ABB RobotStudio station: burguerBotVentosaYCintaDef2.rspag

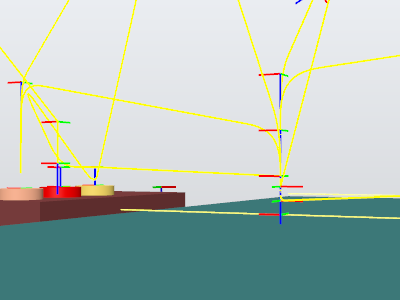
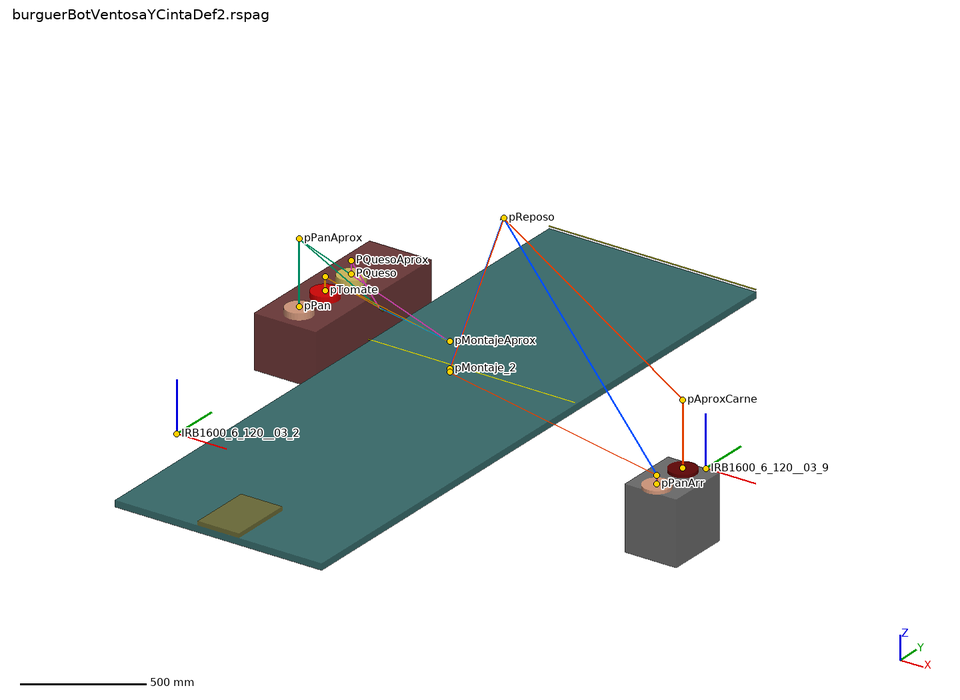
[picture v1: parts stored in the station drawn from their meshes, with robot base, taught points and paths (robot models come from the ABB library and are not in the file)]
--- station ---
Station Station (saved by RobotStudio 24.1.10713.1)
Controller Controlador2, task T_ROB1: task frame (RAPID world) sits at (2496.48, 947.06, 0) mm, rotated rx 0 ry 0 rz 179.92 deg in the station
Controller Controlador4, task T_ROB1: task frame (RAPID world) sits at (600, 0, 0) mm in the station
Controller Controlador4
  mechanical unit ROB_1: IRB1600_6_120__03_2, 6 joints, base frame (0, 0, 0) mm
Controller Controlador2
  mechanical unit ROB_1: IRB1600_6_120__03_9, 6 joints, base frame (0, 0, 0) mm
Layout (positions relative to the parent item):
  - Ventosa [mechanism, from Libraries\Ventosa.rslib] at (1406.29, 0, 929) mm, rotated rx 180 ry 60 rz 180 deg
  - CintaTransportadora [part] at (0, 0, -530) mm, size 1000 x 3000 x 30 mm
  - IRB1600_6_120__03_2 [mechanism, from %ABB.RobotStudio.Models.IRB1600%\IRB1600_6_120_G_03.rslib] at (600, 0, 0) mm; joint values [0, 0, 0, 0, 0.5236, 0] (rad or m)
  - SmartComponent_2 [smart component]
      signals: DO PiezaDetectada, DI ActivaVentosa, DO Vacuostato
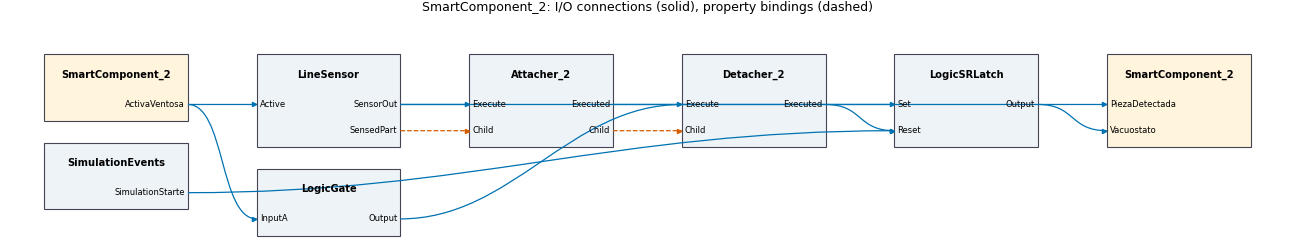
      connections:
        SmartComponent_2.ActivaVentosa -> LineSensor.Active
        SmartComponent_2.ActivaVentosa -> LogicGate.InputA
        LogicGate.Output -> Detacher_2.Execute
        LineSensor.SensorOut -> Attacher_2.Execute
        LineSensor.SensorOut -> SmartComponent_2.PiezaDetectada
        Attacher_2.Executed -> LogicSRLatch.Set
        Detacher_2.Executed -> LogicSRLatch.Reset
        SimulationEvents.SimulationStarted -> LogicSRLatch.Reset
        LogicSRLatch.Output -> SmartComponent_2.Vacuostato
        Attacher_2.Child => Detacher_2.Child
        LineSensor.SensedPart => Attacher_2.Child
    - LineSensor [smart component, from Components\LineSensor.rslib] at (1579.5, 0, 829) mm, rotated rx 180 ry 60 rz 180 deg
        properties: Start=[0 0 -0.002]; End=[0 0 0.02]; Length=0.022; Radius=0.002; Tag=(none); SensedPart=(none); SensedPoint=[0 0 0]
      - _sensorPart_ [part], size 4 x 4 x 22 mm
    - SimulationEvents [smart component, from Components\SimulationEvents.rslib]
    - LogicSRLatch [smart component, from Components\LogicSRLatch.rslib]
    - Attacher_2 [smart component, from Components\Attacher.rslib]
        properties: Parent=Ventosa; Flange=0; Child=(none); Mount=false; Offset=[0 0 0]; Orientation=[0 0 0]
    - Detacher_2 [smart component, from Components\Detacher.rslib]
        properties: Child=(none); KeepPosition=true
    - LogicGate [smart component, from Components\LogicGate.rslib]
        properties: Operator=NOT; Delay=0
  - Pieza_3 [part], size 1050 x 3000 x 100 mm
  - Pieza_7 [part] at (0, -1450, -30) mm, size 200 x 300 x 20 mm
  - SmartComponent_3 [smart component] at (0, 0, -530) mm
      signals: DI PideNuevaPieza, DI MueveCinta, DI Desencolar, DO Hamburguesa_detectada
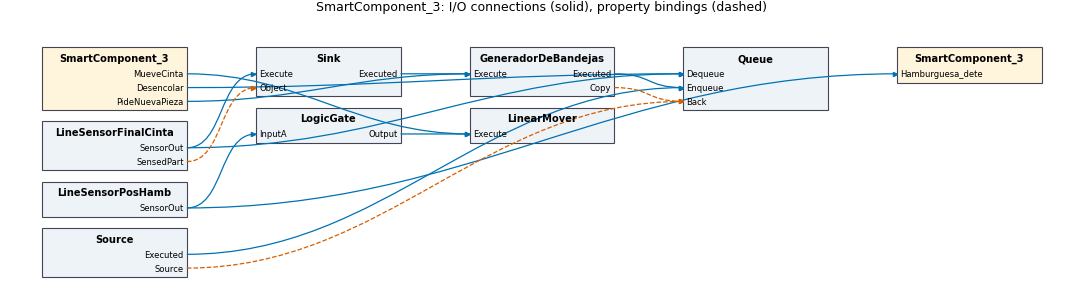
      connections:
        SmartComponent_3.MueveCinta -> LinearMover.Execute
        SmartComponent_3.Desencolar -> Queue.Dequeue
        SmartComponent_3.PideNuevaPieza -> GeneradorDeBandejas.Execute
        GeneradorDeBandejas.Executed -> Queue.Enqueue
        Sink.Executed -> GeneradorDeBandejas.Execute
        LineSensorFinalCinta.SensorOut -> Sink.Execute
        LineSensorFinalCinta.SensorOut -> Queue.Dequeue
        LineSensorPosHamb.SensorOut -> LogicGate.InputA
        LogicGate.Output -> LinearMover.Execute
        LineSensorPosHamb.SensorOut -> SmartComponent_3.Hamburguesa_detectada
        Source.Executed -> Queue.Enqueue
        GeneradorDeBandejas.Copy => Queue.Back
        LineSensorFinalCinta.SensedPart => Sink.Object
        Source.Source => Queue.Back
    - GeneradorDeBandejas [smart component, from Components\Source.rslib]
        properties: Source=Pieza_7; Copy=(none); Parent=(none); Position=[0 -1.45 -0.03]; Orientation=[0 0 0]; Transient=false; PhysicsBehavior=-1
    - LinearMover [smart component, from Components\LinearMover.rslib]
        properties: Object=Queue; Direction=[0 1 0]; Speed=0.2; Reference=Global; ReferenceObject=(none)
    - Queue [smart component, from Components\Queue.rslib]
        properties: Back=(none); Front=(none); Queue={1fa18e9d-088c-41fe-8e63-321db63f1bad};{66fc0b19-5291-4fa8-960b-30c1fd8ad654};{bf5ac1da-f569-4681-bc2f-d1bebfeb1945};{a7c02364-1145-4610-8c2b-21e8e4e74e7e};{e07134d1-5b8f-4729-998b-d35f37be9415};{77c18e64-ed22-4101-8412-22759ad2fd65};{e3f1d31c-383c-4d57-a647-59baedf5051e};{31de0638-30c3-4a0d-b96c-771df3fa9e8e};{ccf4f79c-bd7e-444b-aa3a-f3a101a5e061};{9c3ce438-0d0a-462d-859f-6c1952ce2779};{2c210c3e-426b-4bc3-92f0-a2b14ac0cff1};{860f6b89-5f7b-417f-be90-2e5516634339};{3c4b279c-e194-41e7-8d5b-6c695006562c};{9a04805c-3299-4768-adf6-effe421ff297};{2ba32a07-e99c-497b-b6b1-776f4c664f37};{e5d152f1-81eb-4789-a107-4ce79efd876e};{84050f51-b700-43f5-9d48-1de7078c80f2};{da5c4f3e-e2de-4859-8c8b-22e5639c2eb3};{b8627b52-6deb-4d66-bbe9-42a0777c5345};{afe129ed-1453-4d5a-b210-b8758cc1c2e1};{660fbeab-b469-451a-a4fe-b26f68304c6b};{d46f86e2-3b48-4b92-a915-6ed2dcae6b65};{75fa054e-13a5-4b2b-a626-0fa9227d0997};{dc2c9636-b798-4d71-ba5e-8e763e159b99};{52b1206f-a2cb-4ff9-8ba0-982d9823dc0e};{f684843b-9464-44eb-8d71-6faa8fd13188};{26aecd76-d99c-4597-b4e3-adbf34ae068a};{1ac82643-5105-46b1-9dd2-ef4d0df968c2}; NumberOfObjects=2
    - Sink [smart component, from Components\Sink.rslib]
        properties: Object=(none)
    - LineSensorFinalCinta [smart component, from Components\LineSensor.rslib]
        properties: Start=[2 2 0.76]; End=[1 2 0.76]; Length=1; Radius=0.002; Tag=(none); SensedPart=(none); SensedPoint=[0 0 0]
      - _sensorPart_ [part], size 1000 x 4 x 4 mm
    - LineSensorPosHamb [smart component, from Components\LineSensor.rslib]
        properties: Start=[2 0.75 0.76]; End=[1 0.75 0.76]; Length=1; Radius=0.002; Tag=(none); SensedPart=(none); SensedPoint=[0 0 0]
      - _sensorPart_ [part], size 1000 x 4 x 4 mm
    - LogicGate [smart component, from Components\LogicGate.rslib]
        properties: Operator=NOT; Delay=0
    - Source [smart component, from Components\Source.rslib]
        properties: Source=Pan2; Copy=(none); Parent=(none); Position=[0 0 0]; Orientation=[0 0 0]; Transient=false; PhysicsBehavior=-1
  - Ventosa_2 [mechanism, from Libraries\Ventosa.rslib] at (1690.19, 948.21, 929) mm, rotated rx -180 ry 60 rz -0.08 deg
  - SmartComponent_4 [smart component]
      signals: DO PiezaDetectada, DO Vacuostato, DI ActivaVentosa2
      connections:
        LogicGate.Output -> Detacher_2.Execute
        LineSensor.SensorOut -> Attacher_2.Execute
        LineSensor.SensorOut -> SmartComponent_4.PiezaDetectada
        Attacher_2.Executed -> LogicSRLatch.Set
        Detacher_2.Executed -> LogicSRLatch.Reset
        SimulationEvents.SimulationStarted -> LogicSRLatch.Reset
        LogicSRLatch.Output -> SmartComponent_4.Vacuostato
        SmartComponent_4.ActivaVentosa2 -> LineSensor.Active
        SmartComponent_4.ActivaVentosa2 -> LogicGate.InputA
        Attacher_2.Child => Detacher_2.Child
        LineSensor.SensedPart => Attacher_2.Child
    - LineSensor [smart component, from Components\LineSensor.rslib] at (1516.99, 948.46, 829) mm, rotated rx -180 ry 60 rz -0.08 deg
        properties: Start=[0 0 -0.002]; End=[0 0 0.02]; Length=0.022; Radius=0.002; Tag=(none); SensedPart=(none); SensedPoint=[0 0 0]
      - _sensorPart_ [part], size 4 x 4 x 22 mm
    - SimulationEvents [smart component, from Components\SimulationEvents.rslib]
    - LogicSRLatch [smart component, from Components\LogicSRLatch.rslib]
    - Attacher_2 [smart component, from Components\Attacher.rslib]
        properties: Parent=Ventosa_2; Flange=0; Child=(none); Mount=false; Offset=[0 0 0]; Orientation=[0 0 0]
    - Detacher_2 [smart component, from Components\Detacher.rslib]
        properties: Child=(none); KeepPosition=true
    - LogicGate [smart component, from Components\LogicGate.rslib]
        properties: Operator=NOT; Delay=0
  - Pieza_11 [part], size 304.8 x 406.3 x 254 mm
  - Pieza_12 [part], size 125 x 124.3 x 30 mm
  - Pieza_14 [part], size 250 x 300 x 300 mm
  - Pieza_15 [part] at (0, 75, 0) mm, size 125 x 124.3 x 15 mm
  - IRB1600_6_120__03_9 [mechanism, from %ABB.RobotStudio.Models.IRB1600%\IRB1600_6_120_G_03.rslib] at (2496.48, 947.06, 0) mm, rotated rx 0 ry 0 rz 179.92 deg; joint values [0, 0, 0, 0, 0.5236, 0] (rad or m)
  - Tomate [part] at (0, 180, 0) mm, size 125 x 124.3 x 30 mm
  - Queso [part] at (0, 360, 0) mm, size 125 x 124.3 x 30 mm
  - Pan2 [part] at (0, -105, 0) mm, size 125 x 124.3 x 15 mm
  - Pieza_18 [part] at (0, 400, 0) mm, size 300 x 400 x 250 mm
  - Pieza_7_11 [part] at (0, -1450, -30) mm, size 200 x 300 x 20 mm
  - Pieza_7_51 [part] at (0, -1450, -30) mm, size 200 x 300 x 20 mm
  - Pieza_7_54 [part] at (0, -1450, -30) mm, size 200 x 300 x 20 mm
  - Pieza_7_2 [part] at (0, -1450, -30) mm, size 200 x 300 x 20 mm
Attachment: Ventosa is attached to IRB1600_6_120__03_2 / Link6
Attachment: LineSensor is attached to Ventosa / PiezaVentosa
Attachment: SmartComponent_3 is attached to CintaTransportadora
Attachment: LineSensor is attached to Ventosa_2 / PiezaVentosa
Attachment: Ventosa_2 is attached to IRB1600_6_120__03_9 / Link6
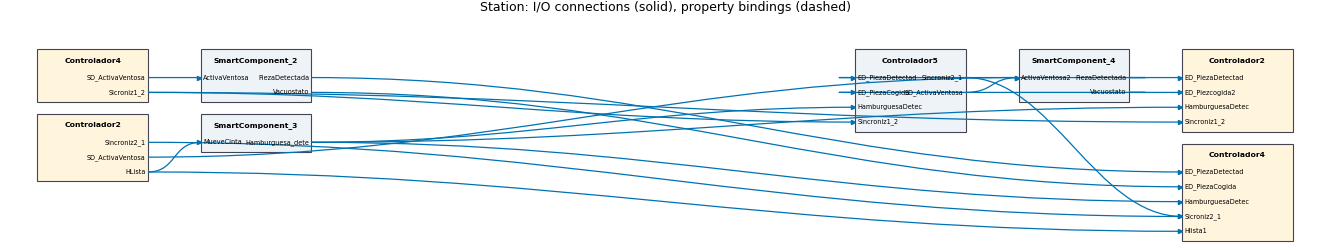
Station logic (signal -> signal, property => property):
  SmartComponent_2.PiezaDetectada -> Controlador4.ED_PiezaDetectada
  Controlador4.SD_ActivaVentosa -> SmartComponent_2.ActivaVentosa
  SmartComponent_2.Vacuostato -> Controlador4.ED_PiezaCogida
  SmartComponent_3.Hamburguesa_detectada -> Controlador4.HamburguesaDetect
  SmartComponent_4.PiezaDetectada -> Controlador5.ED_PiezaDetectada
  SmartComponent_4.Vacuostato -> Controlador5.ED_PiezaCogida
  SmartComponent_3.Hamburguesa_detectada -> Controlador5.HamburguesaDetect
  Controlador5.Sincroniz2_1 -> Controlador4.Sicroniz2_1
  Controlador4.Sicroniz1_2 -> Controlador5.Sincroniz1_2
  SmartComponent_4.PiezaDetectada -> Controlador2.ED_PiezaDetectada2
  SmartComponent_4.Vacuostato -> Controlador2.ED_Piezcogida2
  SmartComponent_3.Hamburguesa_detectada -> Controlador2.HamburguesaDetect2
  Controlador4.Sicroniz1_2 -> Controlador2.Sincroniz1_2
  Controlador2.Sincroniz2_1 -> Controlador4.Sicroniz2_1
  ?.SD_ActivaVentosa -> SmartComponent_4.ActivaVentosa2
  Controlador2.SD_ActivaVentosa -> SmartComponent_4.ActivaVentosa2
  Controlador2.HLista -> SmartComponent_3.MueveCinta
  Controlador2.HLista -> Controlador4.Hlista1

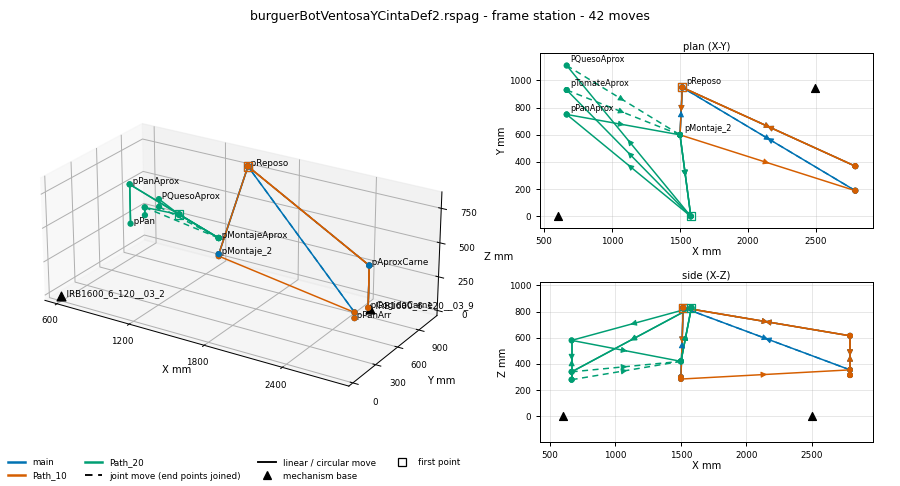
[picture p0: tool path of burguerBotVentosaYCintaDef2.rspag in frame station, 42 of 47 moves have a stored position in this frame; points joined in program order, loops and branches not executed]
--- Backups/Controlador2/RAPID/TASK1/PROGMOD/CalibData.mod ---
MODULE CalibData
    PERS tooldata Ventosa:=[TRUE,[[0,0,200],[1,0,0,0]],[1,[0,0,125],[1,0,0,0],0.002,0.002,0.0013]];
ENDMODULE

--- Backups/Controlador2/RAPID/TASK1/PROGMOD/Module1.mod ---
MODULE Module1
    CONST robtarget pReposo:=[[979.496732003,0,829],[0.5,0,0.866025404,0],[0,0,-1,0],[9E+09,9E+09,9E+09,9E+09,9E+09,9E+09]];
    CONST robtarget pAproxCarne:=[[-294.1282673,577.734595344,615],[0,0.999999744,0.000716141,0],[1,0,1,0],[9E+09,9E+09,9E+09,9E+09,9E+09,9E+09]];
    CONST robtarget pCogidaCarne:=[[-294.1282673,577.734595344,315],[0,0.999999744,0.000716141,0],[1,0,1,0],[9E+09,9E+09,9E+09,9E+09,9E+09,9E+09]];
    CONST robtarget pMontaje_2:=[[995.982835611,348.8831626,300],[0,-0.000716141,0.999999744,0],[0,0,0,0],[9E+09,9E+09,9E+09,9E+09,9E+09,9E+09]];
    CONST robtarget pMontaje:=[[995.982835611,348.8831626,285],[0,-0.000716141,0.999999744,0],[0,0,0,0],[9E+09,9E+09,9E+09,9E+09,9E+09,9E+09]];
    CONST robtarget pPanArr_2:=[[-294.386077932,757.734410716,355],[0,0.999999744,0.000716141,0],[1,0,-1,0],[9E+09,9E+09,9E+09,9E+09,9E+09,9E+09]];
    CONST robtarget pPanArr:=[[-294.386077932,757.734410716,315],[0,0.999999744,0.000716141,0],[1,0,-1,0],[9E+09,9E+09,9E+09,9E+09,9E+09,9E+09]];
!***********************************************************
    !
    ! M?dulo:  Module1
    !
    ! Descripción:
    !   <Introduzca la descripción aquí>
    !
    ! Autor: rafac
    !
    ! Versión: 1.0
    !
    !***********************************************************


    !***********************************************************
    !
    ! Procedimiento Main
    !
    !   Este es el punto de entrada de su programa
    !
    !***********************************************************
    PROC main()
        VAR robtarget aux;
        SetDO Sincroniz2_1,0;
        SetDO HLista, 0;
         WaitDI Sincroniz1_2,1;
            MoveL pReposo,v1000,z100,Ventosa\WObj:=wobj0;
            MoveJ pAproxCarne,v1000,fine,Ventosa\WObj:=wobj0;
            MoveL pCogidaCarne,v500,fine,Ventosa\WObj:=wobj0;
            SetDO SD_ActivaVentosa,1;
            WaitDI ED_Piezcogida2,1;

            MoveL pAproxCarne,v1000,fine,Ventosa\WObj:=wobj0;
            MoveJ pReposo,v1000,fine,Ventosa\WObj:=wobj0;

            MoveL pMontaje_2,v1000,fine,Ventosa\WObj:=wobj0;
            MoveL pMontaje,v1000,fine,Ventosa\WObj:=wobj0;

            SetDO SD_ActivaVentosa,0;
            WaitDI ED_Piezcogida2,0;

            MoveL pMontaje_2,v1000,fine,Ventosa\WObj:=wobj0;
            MoveL pReposo,v1000,z100,Ventosa\WObj:=wobj0;
            SetDO HLista, 1;

            SetDO Sincroniz2_1,1;
            WaitDI Sincroniz1_2, 1;

            MoveL pPanArr_2,v1000,fine,Ventosa\WObj:=wobj0;
            MoveL pPanArr,v1000,fine,Ventosa\WObj:=wobj0;

            SetDO SD_ActivaVentosa,1;
            WaitDI ED_Piezcogida2,1;

            MoveL pPanArr_2,v1000,fine,Ventosa\WObj:=wobj0;
            MoveJ pReposo,v1000,fine,Ventosa\WObj:=wobj0;

            aux := Offs(pMontaje, 0, 0,45);

            MoveL aux,v1000,fine,Ventosa\WObj:=wobj0;


            SetDO SD_ActivaVentosa,0;
            WaitDI ED_Piezcogida2,0;

            aux := Offs(pMontaje, 0, 0, 54);

            MoveL aux,v1000,fine,Ventosa\WObj:=wobj0;
            MoveL pReposo,v1000,z100,Ventosa\WObj:=wobj0;
            SetDO Sincroniz2_1,0;


    ENDPROC
    PROC Path_10()
        MoveL pReposo,v1000,z100,Ventosa\WObj:=wobj0;
        MoveL pAproxCarne,v1000,z100,Ventosa\WObj:=wobj0;
        MoveL pCogidaCarne,v1000,z100,Ventosa\WObj:=wobj0;
        MoveL pAproxCarne,v1000,z100,Ventosa\WObj:=wobj0;
        MoveL pReposo,v1000,z100,Ventosa\WObj:=wobj0;
        MoveL pMontaje_2,v1000,z100,Ventosa\WObj:=wobj0;
        MoveL pMontaje,v1000,z100,Ventosa\WObj:=wobj0;
        MoveL pPanArr_2,v1000,z100,Ventosa\WObj:=wobj0;
        MoveL pPanArr,v1000,z100,Ventosa\WObj:=wobj0;

    ENDPROC
ENDMODULE

--- Backups/Controlador4/RAPID/TASK1/PROGMOD/CalibData.mod ---
MODULE CalibData
    PERS tooldata Ventosa:=[TRUE,[[0,0,200],[1,0,0,0]],[1,[0,0,125],[1,0,0,0],0.002,0.002,0.0013]];
    TASK PERS wobjdata Workobject_1:=[FALSE,TRUE,"",[[400,2000,250],[0,1,0,0]],[[0,0,0],[1,0,0,0]]];
ENDMODULE

--- Backups/Controlador4/RAPID/TASK1/PROGMOD/Module1.mod ---
MODULE Module1
    CONST robtarget pReposo:=[[979.496732003,0,829],[0.5,0,0.866025404,0],[0,0,-1,0],[9E+09,9E+09,9E+09,9E+09,9E+09,9E+09]];
    CONST robtarget pAprox:=[[550,1450,-200],[0,0,0,1],[0,0,0,0],[9E+09,9E+09,9E+09,9E+09,9E+09,9E+09]];
    CONST robtarget pCogida:=[[550,1450,-100],[0,0,0,1],[0,0,0,0],[9E+09,9E+09,9E+09,9E+09,9E+09,9E+09]];
    CONST robtarget pMontajeAprox:=[[900,599.6,420],[0,0,1,0],[0,0,0,0],[9E+09,9E+09,9E+09,9E+09,9E+09,9E+09]];
    CONST robtarget pMontaje:=[[900,599.6,240],[0,0,1,0],[0,0,0,0],[9E+09,9E+09,9E+09,9E+09,9E+09,9E+09]];
    CONST robtarget pPanAprox:=[[66.288,749.687,580],[0,0,1,0],[0,0,0,0],[9E+09,9E+09,9E+09,9E+09,9E+09,9E+09]];
    CONST robtarget pPan:=[[66.288,749.687,280],[0,0,1,0],[0,0,0,0],[9E+09,9E+09,9E+09,9E+09,9E+09,9E+09]];
    CONST robtarget pCarne:=[[2189.782,368.901,315],[0,0,1,0],[0,0,0,0],[9E+09,9E+09,9E+09,9E+09,9E+09,9E+09]];
    CONST robtarget pCarneAprox:=[[2189.782,368.901,615],[0,0,1,0],[0,0,0,0],[9E+09,9E+09,9E+09,9E+09,9E+09,9E+09]];
    CONST robtarget PQueso:=[[66.288,1109.687,280],[0,0,1,0],[0,0,0,0],[9E+09,9E+09,9E+09,9E+09,9E+09,9E+09]];
    CONST robtarget pTomateAprox:=[[66.288,929.687,340],[0,0,1,0],[0,0,0,0],[9E+09,9E+09,9E+09,9E+09,9E+09,9E+09]];
    CONST robtarget pTomate:=[[66.288,929.687,280],[0,0,1,0],[0,0,0,0],[9E+09,9E+09,9E+09,9E+09,9E+09,9E+09]];
    CONST robtarget PQuesoAprox:=[[66.288,1109.687,340],[0,0,1,0],[0,0,0,0],[9E+09,9E+09,9E+09,9E+09,9E+09,9E+09]];
    CONST robtarget pMon2:=[[900,599.6,322],[0,0,1,0],[0,-2,1,2],[9E+09,9E+09,9E+09,9E+09,9E+09,9E+09]];
!***********************************************************
    !
    ! M?dulo:  Module1
    !
    ! Descripción:
    !   <Introduzca la descripción aquí>
    !
    ! Autor: rafac
    !
    ! Versión: 1.0
    !
    !***********************************************************


    !***********************************************************
    !
    ! Procedimiento Main
    !
    !   Este es el punto de entrada de su programa
    !
    !***********************************************************
    PROC main()
        Path_20;

    ENDPROC

    PROC Path_20()

                         VAR robtarget aux;
        SetDO Sicroniz1_2,0;

        aux:=Offs(pMontaje,0,0,30);
            WaitDI HamburguesaDetect,1;
           WaitDi Hlista1,0;
            MoveL pReposo,v1000,z100,Ventosa\WObj:=wobj0;
            MoveL pPanAprox,v1000,fine,Ventosa\WObj:=wobj0;
            MoveL pPan,v1000,fine,Ventosa\WObj:=wobj0;
            SetDO SD_ActivaVentosa,1;
            WaitDI ED_PiezaCogida,1;

            MoveL pPanAprox,v1000,fine,Ventosa\WObj:=wobj0;
            MoveL pMontajeAprox,v1000,fine,Ventosa\WObj:=wobj0;

            MoveL aux,v1000,fine,Ventosa\WObj:=wobj0;

            SetDO SD_ActivaVentosa,0;
            WaitDI ED_PiezaCogida,0;

            MoveL pMontajeAprox,v1000,fine,Ventosa\WObj:=wobj0;
            MoveL pReposo,v1000,z100,Ventosa\WObj:=wobj0;

            SetDO Sicroniz1_2,1;
            SetDO Sicroniz1_2,0;
            WaitDI Sicroniz2_1, 1;


            IF HQueso = 1 THEN
                MoveL PQuesoAprox,v1000,fine,Ventosa\WObj:=wobj0;
                MoveL PQueso,v1000,fine,Ventosa\WObj:=wobj0;

                SetDO SD_ActivaVentosa,1;
                WaitDI ED_PiezaCogida,1;

                MoveJ pMontajeAprox,v500,fine,Ventosa\WObj:=wobj0;

                MoveL Offs(aux,0,0,45),v100,fine,Ventosa\WObj:=wobj0;

                SetDO SD_ActivaVentosa,0;
                WaitDI ED_PiezaCogida,0;

                MoveL pMontajeAprox,v1000,fine,Ventosa\WObj:=wobj0;
                MoveL pReposo,v1000,z100,Ventosa\WObj:=wobj0;
            ELSE

                MoveL pTomateAprox,v1000,fine,Ventosa\WObj:=wobj0;
                MoveL pTomate,v1000,fine,Ventosa\WObj:=wobj0;

                SetDO SD_ActivaVentosa,1;
                WaitDI ED_PiezaCogida,1;

                MoveL pTomateAprox,v1000,fine,Ventosa\WObj:=wobj0;
                MoveJ pMontajeAprox,v500,fine,Ventosa\WObj:=wobj0;
                MoveL Offs(aux,0,0,45),v100,fine,Ventosa\WObj:=wobj0;

                SetDO SD_ActivaVentosa,0;
                WaitDI ED_PiezaCogida,0;

                MoveL pMontajeAprox,v1000,fine,Ventosa\WObj:=wobj0;
                MoveL pReposo,v1000,z100,Ventosa\WObj:=wobj0;

            ENDIF
            MoveL pReposo,v1000,z100,Ventosa\WObj:=wobj0;

            SetDO Sicroniz1_2,1;


    ENDPROC
ENDMODULE

--- Backups/Controlador2/SYSPAR/EIO.cfg ---
EIO:CFG_1.0:6:1::
#
INDUSTRIAL_NETWORK:

      -Name "DeviceNet" -Label "DeviceNet Master/Slave Network" -Address "2"
#
DEVICENET_DEVICE:

      -Name "MiDeviceNet"
#
DEVICENET_INTERNAL_DEVICE:

      -Name "DN_Internal_Device" -VendorName "ABB Robotics"\
      -ProductName "DeviceNet Internal Slave Device"
#
EIO_SIGNAL:

      -Name "ED_Piezcogida2" -SignalType "DI" -Device "MiDeviceNet"\
      -Label "ED_Piezcogida2" -DeviceMap "1" -Access "All"

      -Name "ED_PiezaDetectada2" -SignalType "DI" -Device "MiDeviceNet"\
      -Label "ED_PiezaDetectada2" -DeviceMap "2" -Access "All"

      -Name "HamburguesaDetect2" -SignalType "DI" -Device "MiDeviceNet"\
      -Label "HamburguesaDetect2" -DeviceMap "3" -Access "All"

      -Name "Sincroniz1_2" -SignalType "DI" -Device "MiDeviceNet"\
      -Label "Sincroniz1_2" -DeviceMap "4" -Access "All"

      -Name "Sincroniz2_1" -SignalType "DO" -Device "MiDeviceNet"\
      -Label "Sincroniz2_1" -DeviceMap "2" -Access "All"

      -Name "SD_ActivaVentosa" -SignalType "DO" -Device "MiDeviceNet"\
      -Label "SD_ActivaVentosa" -DeviceMap "3" -Access "All"

      -Name "HLista" -SignalType "DO" -Device "MiDeviceNet" -Label "HLista"\
      -DeviceMap "6" -Access "All"

--- Backups/Controlador4/SYSPAR/EIO.cfg ---
EIO:CFG_1.0:6:1::
#
INDUSTRIAL_NETWORK:

      -Name "DeviceNet" -Label "DeviceNet Master/Slave Network" -Address "2"
#
DEVICENET_DEVICE:

      -Name "MiDeviceNet"
#
DEVICENET_INTERNAL_DEVICE:

      -Name "DN_Internal_Device" -VendorName "ABB Robotics"\
      -ProductName "DeviceNet Internal Slave Device"
#
EIO_SIGNAL:

      -Name "ED_PiezaDetectada" -SignalType "DI" -Device "MiDeviceNet"\
      -Label "ED_PiezaDetectada" -DeviceMap "0" -Access "All"

      -Name "ED_PiezaCogida" -SignalType "DI" -Device "MiDeviceNet"\
      -Label "ED_PiezaCogida" -DeviceMap "1" -Access "All"

      -Name "SD_ActivaVentosa" -SignalType "DO" -Device "MiDeviceNet"\
      -Label "SD_ActivaVentosa" -DeviceMap "0" -Access "All"

      -Name "HamburguesaDetect" -SignalType "DI" -Device "MiDeviceNet"\
      -Label "HamburguesaDetect" -DeviceMap "3" -Access "All"

      -Name "Sicroniz2_1" -SignalType "DI" -Device "MiDeviceNet"\
      -Label "Sicroniz2_1" -DeviceMap "4" -Access "All"

      -Name "Sicroniz1_2" -SignalType "DO" -Device "MiDeviceNet"\
      -Label "Sicroniz1_2" -DeviceMap "3" -Access "All"

      -Name "HQueso" -SignalType "DI" -Device "MiDeviceNet" -DeviceMap "2"\
      -Access "All"

      -Name "Hlista1" -SignalType "DI" -Device "MiDeviceNet" -Label "Hlista1"\
      -DeviceMap "5"

      -Name "cogePan" -SignalType "DO" -Device "MiDeviceNet" -Label "cogePan"\
      -DeviceMap "6"
